(* Schneider Machine Expert - Basic project Motor_StartStop_Overload_TM221CE16T, file version 3.0.0.0 *)
(* ProjectInformations: Name=New project *)

HARDWARE
  Cpu 0: TM221CE16T
  EthernetConfiguration: NetworkName=M221, IpAllocationMode=FixedAddress, IpAddress=0.0.0.0, SubnetMask=0.0.0.0
  SerialLineConfiguration: Baud=Baud19200, Parity=ParityEven, DataBits=DataBits8, StopBits=StopBits1, PhysicalMedium=PhysicalMediumRs485, TransmissionMode=TransmissionModeModbusRtu, SlaveId=1, Addressing=SlaveAddressing
  MastTask: UsePeriodScanMode=false, PeriodScan=100
  FastTask: Period=255
  CpuBehavior: StartingMode=StartAsPreviousState, AutoSaveRamOnEeprom=true, WatchdogPeriod=250

SYMBOLS  (address, symbol, comment, settings)
  %M0       SYSTEM_READY
  %M1       MOTOR_RUNNING
  %M2       OVERLOAD_ALARM
  %M3       ANY_ALARM
  %TM0        [Preset=3, Base=OneSecond]
  %TM1        [Preset=5, Base=HundredMilliseconds]
  %I0.0     EMERGENCY_PB

POU Motor_Control
  (* SectionNumber=0 *)

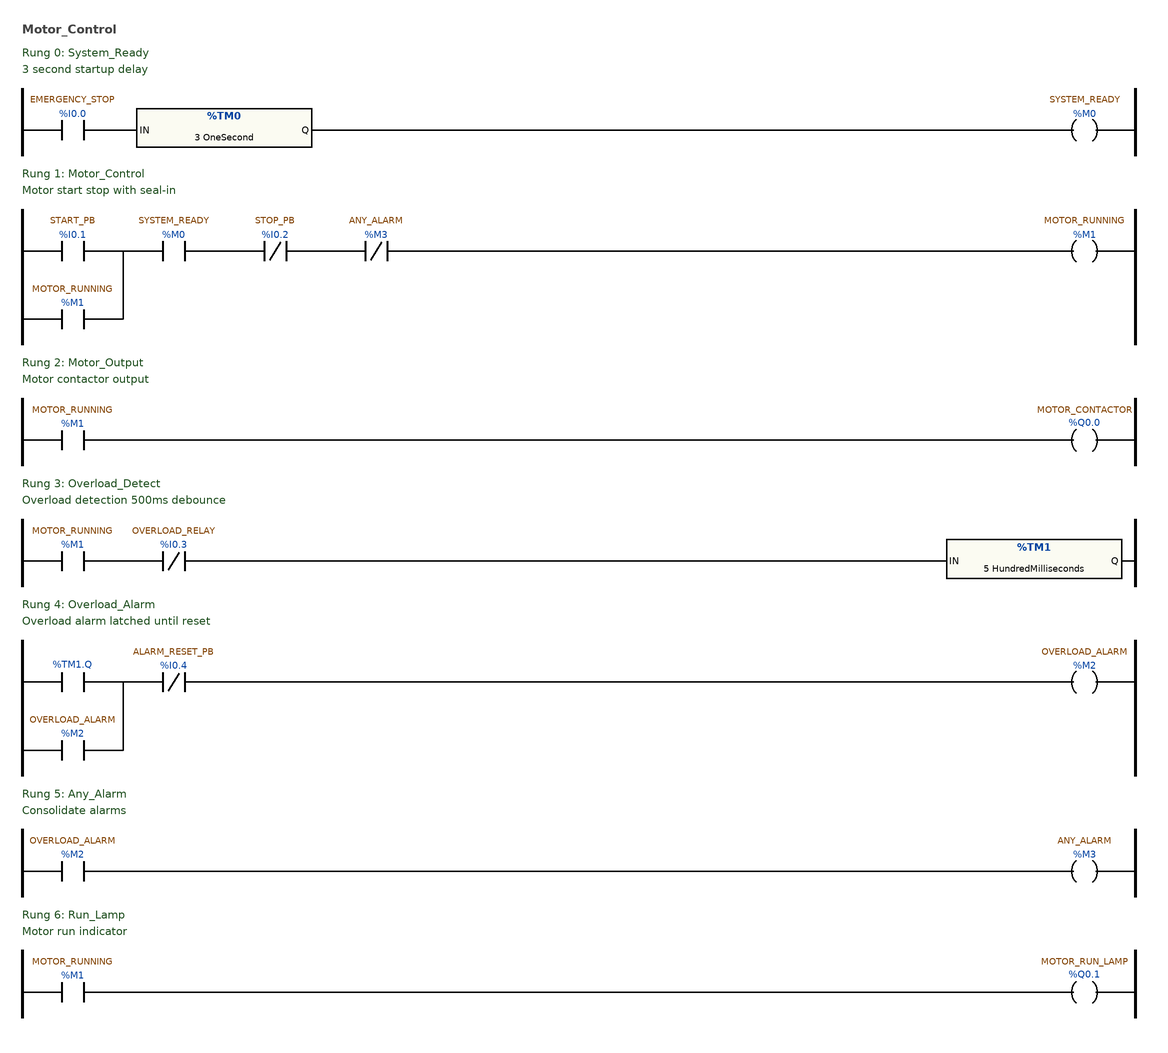

// Rung 0: System_Ready
// 3 second startup delay
  BLK %TM0
  LD %I0.0                (* EMERGENCY_PB *)
  IN
  OUT_BLK
  LD Q
  ST %M0                  (* SYSTEM_READY *)
  END_BLK
  // %I0.0: Emergency Stop OK
  // %M0: System Ready
  // as ST:
  //   %TM0(IN := EMERGENCY_PB);
  //   SYSTEM_READY := %TM0.Q;

// Rung 1: Motor_Control
// Motor start stop with seal-in
  LD %I0.1
  OR %M1                  (* MOTOR_RUNNING *)
  AND %M0                 (* SYSTEM_READY *)
  ANDN %I0.2
  ANDN %M3                (* ANY_ALARM *)
  ST %M1                  (* MOTOR_RUNNING *)
  // %I0.1: Start PB
  // %I0.2: Stop NC
  // %M3: No Alarm
  // %M1: Motor Run
  // %M1: Seal-In
  // as ST:
  //   MOTOR_RUNNING := (%I0.1 OR MOTOR_RUNNING) AND SYSTEM_READY AND NOT %I0.2 AND NOT ANY_ALARM;

// Rung 2: Motor_Output
// Motor contactor output
  LD %M1                  (* MOTOR_RUNNING *)
  ST %Q0.0
  // %Q0.0: Motor Output
  // as ST:
  //   %Q0.0 := MOTOR_RUNNING;

// Rung 3: Overload_Detect
// Overload detection 500ms debounce
  BLK %TM1
  LD %M1                  (* MOTOR_RUNNING *)
  ANDN %I0.3
  IN
  OUT_BLK
  END_BLK
  // %I0.3: OL Trip NC
  // as ST:
  //   %TM1(IN := MOTOR_RUNNING AND NOT %I0.3);

// Rung 4: Overload_Alarm
// Overload alarm latched until reset
  LD %TM1.Q
  OR %M2                  (* OVERLOAD_ALARM *)
  ANDN %I0.4
  ST %M2                  (* OVERLOAD_ALARM *)
  // %TM1.Q: OL Confirm
  // %I0.4: Reset
  // %M2: OL Alarm
  // %M2: Latch
  // as ST:
  //   OVERLOAD_ALARM := (%TM1.Q OR OVERLOAD_ALARM) AND NOT %I0.4;

// Rung 5: Any_Alarm
// Consolidate alarms
  LD %M2                  (* OVERLOAD_ALARM *)
  ST %M3                  (* ANY_ALARM *)
  // %M3: Any Alarm
  // as ST:
  //   ANY_ALARM := OVERLOAD_ALARM;

// Rung 6: Run_Lamp
// Motor run indicator
  LD %M1                  (* MOTOR_RUNNING *)
  ST %Q0.1
  // %Q0.1: Run Lamp
  // as ST:
  //   %Q0.1 := MOTOR_RUNNING;

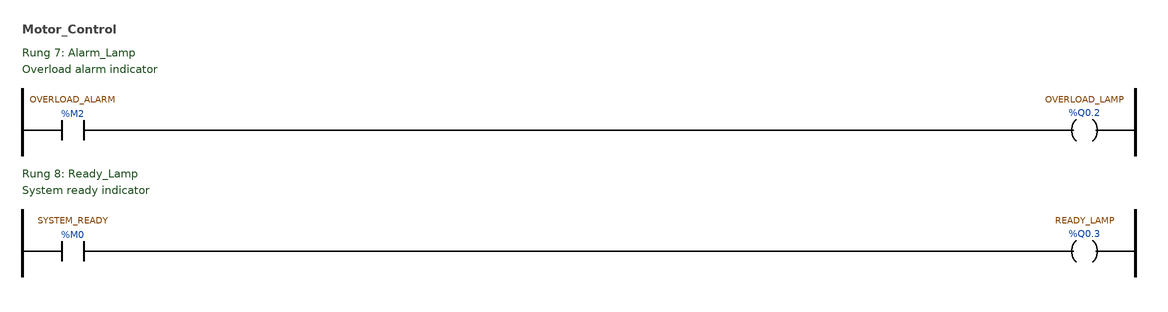

// Rung 7: Alarm_Lamp
// Overload alarm indicator
  LD %M2                  (* OVERLOAD_ALARM *)
  ST %Q0.2
  // %Q0.2: Alarm Lamp
  // as ST:
  //   %Q0.2 := OVERLOAD_ALARM;

// Rung 8: Ready_Lamp
// System ready indicator
  LD %M0                  (* SYSTEM_READY *)
  ST %Q0.3
  // %Q0.3: Ready Lamp
  // as ST:
  //   %Q0.3 := SYSTEM_READY;
